{attribute 'qualified_only'}
{attribute 'strict'}
TYPE E_PIEZO_SUBSTATE :
(
	NONE				:= 0,
	
	NOTOP_NOTREADY		:= 100,
	NOTOP_READY			:= 101,
	NOTOP_ERROR			:= 199,
	
	OP_POS				:= 203,            
	OP_AUTO				:= 204,
	OP_ERROR			:= 299
);
END_TYPE

(* stored: Version 1.1.0.1, ProductVersion 3.1.4022.16
   DUT E_PIEZO_SUBSTATE: Id {799404c9-da36-48d5-9ce1-118394e18490} *)
